PROGRAM MAIN
VAR
END_VAR

END_PROGRAM

(* stored: Version 1.1.0.1
   POU MAIN: Id {a30c69d7-c52a-442a-bd8c-3c5ceebff2cd} *)
